// TIA Portal V20 export
DATA_BLOCK "DB_ConveyorParameters"   // DB7
// stored: Access Published, MemoryReserve 100, Namespace Global
   VAR
      Line : Struct
         ProductionLine : Struct
            Conveyor : Array[_.gminProductionLine.._.gmaxProductionLine] of "Global.ConveyorParameters";
            TransferUnit { S7_SetPoint := 'True'} : Array[_.gminProductionLine.._.gmaxProductionLine] of "Global.ConveyorParameters_TransferUnit";
         END_STRUCT;
         EmptyLine : Struct
            Conveyor : Array[_.gminEmptyLine.._.gmaxEmptyLine] of "Global.ConveyorParameters";
         END_STRUCT;
         PackedLine : Struct
            Conveyor : Array[_.gminPackedLine.._.gmaxPackedLine] of "Global.ConveyorParameters";
         END_STRUCT;
      END_STRUCT;
   END_VAR
BEGIN
END_DATA_BLOCK
